// TIA Portal V17 export
// export: Created 2025-03-05T08:00:07.6306461Z, ExportSetting WithDefaults, DisplayName Totally Integrated Automation Portal, DisplayVersion V17 Update 8, DisplayName TIA Portal Openness, DisplayVersion V17 Update 8, DisplayName TIA Portal Version Control Interface, DisplayVersion V17, DisplayName SINAMICS Startdrive Advanced, DisplayVersion V17 SP2, DisplayName SINAMICS Startdrive G110M, G120, G120C, G120D, G120P, G115D, DisplayVersion V17 SP2, DisplayName SINAMICS Startdrive G130, G150, S120, S150, SINAMICS MV, S210, DisplayVersion V17 SP2, DisplayName STEP 7 Professional, DisplayVersion V17 Update 8, DisplayName SINUMERIK ONE STEP 7 Toolbox, DisplayVersion V17 Update 12, DisplayName SINUMERIK 840D sl STEP 7 Toolbox, DisplayVersion V17 Update 12, DisplayName STEP 7 Safety, DisplayVersion V17 Update 6, DisplayName WinCC Advanced, DisplayVersion V17 Update 8
DATA_BLOCK "DB2031_CYCLES_GENERAL"   // DB2031
{ S7_Optimized_Access := 'FALSE'; DB_Accessible_From_OPC_UA := 'FALSE' }
AUTHOR : ETXETAR
VERSION : 1.0
// stored: AutoNumber false, DBAccessibleFromOPCUA false, DBAccessibleFromWebserver true, IsOnlyStoredInLoadMemory false, IsWriteProtectedInAS false
   VAR RETAIN
      CONTINUOUS_CYCLE { S7_SetPoint := 'True'} : "CYCLES";
      SINGLE_CYCLE { S7_SetPoint := 'True'} : "CYCLES";
      RUN_OUT { S7_SetPoint := 'True'} : "CYCLES";
      DRY_CYCLE { S7_SetPoint := 'True'} : "CYCLES";
      MANUAL_LOAD_CYCLE { S7_SetPoint := 'True'} : "CYCLES";
      GANTRY_ROBOT_TEST_CYCLE { S7_SetPoint := 'True'} : "CYCLES";
      GANTRY_DRY_CYCLE { S7_SetPoint := 'True'} : "CYCLES";
      ROBOT_DRY_CYCLE { S7_SetPoint := 'True'} : "CYCLES";
      CALIBRATION_CYCLE { S7_SetPoint := 'True'} : "CYCLES";
      RUN_OUT_UNIT_01 { S7_SetPoint := 'True'} : "CYCLES";
      RUN_OUT_UNIT_02 { S7_SetPoint := 'True'} : "CYCLES";
      MASTER_MEASUREMENT { S7_SetPoint := 'True'} : "CYCLES";
   END_VAR
BEGIN
   CONTINUOUS_CYCLE.GENERAL_CONDITIONS := FALSE;
   CONTINUOUS_CYCLE.INITIAL_CONDITIONS := FALSE;
   CONTINUOUS_CYCLE.ENABLE_REQUEST := FALSE;
   CONTINUOUS_CYCLE.DISABLE_REQUEST := FALSE;
   CONTINUOUS_CYCLE.TOGGLE_COMMAND_P := FALSE;
   CONTINUOUS_CYCLE.WARNING_GONE := FALSE;
   CONTINUOUS_CYCLE.GENERAL_CONDITIONS_HELP := FALSE;
   CONTINUOUS_CYCLE.INITIAL_CONDITIONS_HELP := FALSE;
   CONTINUOUS_CYCLE.CYCLE_SELECTED := FALSE;   // CONTINUOUS CYCLE SELECTED
   CONTINUOUS_CYCLE.CYCLE_SELECTED_AUX := FALSE;
   CONTINUOUS_CYCLE.CYCLE_COMPLETED := FALSE;   // CONTINUOUS CYCLE COMPLETED
   CONTINUOUS_CYCLE.MACHINE_EMPTY := FALSE;
   CONTINUOUS_CYCLE.MACHINE_EMPTY_MANUAL_LOAD_SELECTED := FALSE;
   CONTINUOUS_CYCLE.MACHINE_EMPTY_WO_MANUAL_LOAD_SELECTED := FALSE;
   CONTINUOUS_CYCLE.RESET_FULL_DEPTH_DRY_CYCLE_DISABLED := FALSE;
   CONTINUOUS_CYCLE.RESET_FULL_DEPTHS_AUX := FALSE;
   CONTINUOUS_CYCLE.CYCLE_SEOC := FALSE;
   CONTINUOUS_CYCLE.CYCLE_IS := FALSE;
   SINGLE_CYCLE.GENERAL_CONDITIONS := TRUE;
   SINGLE_CYCLE.INITIAL_CONDITIONS := TRUE;
   SINGLE_CYCLE.ENABLE_REQUEST := FALSE;
   SINGLE_CYCLE.DISABLE_REQUEST := TRUE;
   SINGLE_CYCLE.TOGGLE_COMMAND_P := FALSE;
   SINGLE_CYCLE.WARNING_GONE := FALSE;
   SINGLE_CYCLE.GENERAL_CONDITIONS_HELP := FALSE;
   SINGLE_CYCLE.INITIAL_CONDITIONS_HELP := FALSE;
   SINGLE_CYCLE.CYCLE_SELECTED := FALSE;   // SINGLE CYCLE SELECTED
   SINGLE_CYCLE.CYCLE_SELECTED_AUX := FALSE;
   SINGLE_CYCLE.CYCLE_COMPLETED := FALSE;   // SINGLE CYCLE COMPLETED
   SINGLE_CYCLE.MACHINE_EMPTY := FALSE;
   SINGLE_CYCLE.MACHINE_EMPTY_MANUAL_LOAD_SELECTED := FALSE;
   SINGLE_CYCLE.MACHINE_EMPTY_WO_MANUAL_LOAD_SELECTED := FALSE;
   SINGLE_CYCLE.RESET_FULL_DEPTH_DRY_CYCLE_DISABLED := FALSE;
   SINGLE_CYCLE.RESET_FULL_DEPTHS_AUX := FALSE;
   SINGLE_CYCLE.CYCLE_SEOC := FALSE;
   SINGLE_CYCLE.CYCLE_IS := FALSE;
   RUN_OUT.GENERAL_CONDITIONS := TRUE;
   RUN_OUT.INITIAL_CONDITIONS := TRUE;
   RUN_OUT.ENABLE_REQUEST := FALSE;
   RUN_OUT.DISABLE_REQUEST := FALSE;
   RUN_OUT.TOGGLE_COMMAND_P := FALSE;
   RUN_OUT.WARNING_GONE := FALSE;
   RUN_OUT.GENERAL_CONDITIONS_HELP := FALSE;
   RUN_OUT.INITIAL_CONDITIONS_HELP := FALSE;
   RUN_OUT.CYCLE_SELECTED := FALSE;   // RUN OUT CYCLE SELECTED
   RUN_OUT.CYCLE_SELECTED_AUX := FALSE;
   RUN_OUT.CYCLE_COMPLETED := FALSE;   // RUN OUT CYCLE COMPLETED
   RUN_OUT.MACHINE_EMPTY := FALSE;
   RUN_OUT.MACHINE_EMPTY_MANUAL_LOAD_SELECTED := FALSE;
   RUN_OUT.MACHINE_EMPTY_WO_MANUAL_LOAD_SELECTED := FALSE;
   RUN_OUT.RESET_FULL_DEPTH_DRY_CYCLE_DISABLED := FALSE;
   RUN_OUT.RESET_FULL_DEPTHS_AUX := FALSE;
   RUN_OUT.CYCLE_SEOC := FALSE;
   RUN_OUT.CYCLE_IS := FALSE;
   DRY_CYCLE.GENERAL_CONDITIONS := FALSE;
   DRY_CYCLE.INITIAL_CONDITIONS := FALSE;
   DRY_CYCLE.ENABLE_REQUEST := FALSE;
   DRY_CYCLE.DISABLE_REQUEST := FALSE;
   DRY_CYCLE.TOGGLE_COMMAND_P := FALSE;
   DRY_CYCLE.WARNING_GONE := FALSE;
   DRY_CYCLE.GENERAL_CONDITIONS_HELP := FALSE;
   DRY_CYCLE.INITIAL_CONDITIONS_HELP := FALSE;
   DRY_CYCLE.CYCLE_SELECTED := FALSE;   // DRY CYCLE SELECTED
   DRY_CYCLE.CYCLE_SELECTED_AUX := FALSE;
   DRY_CYCLE.CYCLE_COMPLETED := FALSE;   // DRY CYCLE COMPLETED
   DRY_CYCLE.MACHINE_EMPTY := FALSE;
   DRY_CYCLE.MACHINE_EMPTY_MANUAL_LOAD_SELECTED := FALSE;
   DRY_CYCLE.MACHINE_EMPTY_WO_MANUAL_LOAD_SELECTED := FALSE;
   DRY_CYCLE.RESET_FULL_DEPTH_DRY_CYCLE_DISABLED := FALSE;
   DRY_CYCLE.RESET_FULL_DEPTHS_AUX := FALSE;
   DRY_CYCLE.CYCLE_SEOC := FALSE;
   DRY_CYCLE.CYCLE_IS := FALSE;
   MANUAL_LOAD_CYCLE.GENERAL_CONDITIONS := FALSE;
   MANUAL_LOAD_CYCLE.INITIAL_CONDITIONS := TRUE;
   MANUAL_LOAD_CYCLE.ENABLE_REQUEST := FALSE;
   MANUAL_LOAD_CYCLE.DISABLE_REQUEST := FALSE;
   MANUAL_LOAD_CYCLE.TOGGLE_COMMAND_P := FALSE;
   MANUAL_LOAD_CYCLE.WARNING_GONE := TRUE;
   MANUAL_LOAD_CYCLE.GENERAL_CONDITIONS_HELP := FALSE;
   MANUAL_LOAD_CYCLE.INITIAL_CONDITIONS_HELP := FALSE;
   MANUAL_LOAD_CYCLE.CYCLE_SELECTED := TRUE;   // MANUAL LOAD CYCLE SELECTED
   MANUAL_LOAD_CYCLE.CYCLE_SELECTED_AUX := FALSE;
   MANUAL_LOAD_CYCLE.CYCLE_COMPLETED := FALSE;   // MANUAL LOAD CYCLE COMPLETED
   MANUAL_LOAD_CYCLE.MACHINE_EMPTY := FALSE;
   MANUAL_LOAD_CYCLE.MACHINE_EMPTY_MANUAL_LOAD_SELECTED := FALSE;
   MANUAL_LOAD_CYCLE.MACHINE_EMPTY_WO_MANUAL_LOAD_SELECTED := FALSE;
   MANUAL_LOAD_CYCLE.RESET_FULL_DEPTH_DRY_CYCLE_DISABLED := FALSE;
   MANUAL_LOAD_CYCLE.RESET_FULL_DEPTHS_AUX := FALSE;
   MANUAL_LOAD_CYCLE.CYCLE_SEOC := FALSE;
   MANUAL_LOAD_CYCLE.CYCLE_IS := FALSE;
   GANTRY_ROBOT_TEST_CYCLE.GENERAL_CONDITIONS := FALSE;
   GANTRY_ROBOT_TEST_CYCLE.INITIAL_CONDITIONS := FALSE;
   GANTRY_ROBOT_TEST_CYCLE.ENABLE_REQUEST := FALSE;
   GANTRY_ROBOT_TEST_CYCLE.DISABLE_REQUEST := FALSE;
   GANTRY_ROBOT_TEST_CYCLE.TOGGLE_COMMAND_P := FALSE;
   GANTRY_ROBOT_TEST_CYCLE.WARNING_GONE := FALSE;
   GANTRY_ROBOT_TEST_CYCLE.GENERAL_CONDITIONS_HELP := FALSE;
   GANTRY_ROBOT_TEST_CYCLE.INITIAL_CONDITIONS_HELP := FALSE;
   GANTRY_ROBOT_TEST_CYCLE.CYCLE_SELECTED := FALSE;   // GANTRY ROBOT TEST CYCLE SELECTED
   GANTRY_ROBOT_TEST_CYCLE.CYCLE_SELECTED_AUX := FALSE;
   GANTRY_ROBOT_TEST_CYCLE.CYCLE_COMPLETED := FALSE;   // GANTRY ROBOT TEST CYCLE COMPLETED
   GANTRY_ROBOT_TEST_CYCLE.MACHINE_EMPTY := FALSE;
   GANTRY_ROBOT_TEST_CYCLE.MACHINE_EMPTY_MANUAL_LOAD_SELECTED := FALSE;
   GANTRY_ROBOT_TEST_CYCLE.MACHINE_EMPTY_WO_MANUAL_LOAD_SELECTED := FALSE;
   GANTRY_ROBOT_TEST_CYCLE.RESET_FULL_DEPTH_DRY_CYCLE_DISABLED := FALSE;
   GANTRY_ROBOT_TEST_CYCLE.RESET_FULL_DEPTHS_AUX := FALSE;
   GANTRY_ROBOT_TEST_CYCLE.CYCLE_SEOC := FALSE;
   GANTRY_ROBOT_TEST_CYCLE.CYCLE_IS := FALSE;
   GANTRY_DRY_CYCLE.GENERAL_CONDITIONS := FALSE;
   GANTRY_DRY_CYCLE.INITIAL_CONDITIONS := FALSE;
   GANTRY_DRY_CYCLE.ENABLE_REQUEST := FALSE;
   GANTRY_DRY_CYCLE.DISABLE_REQUEST := FALSE;
   GANTRY_DRY_CYCLE.TOGGLE_COMMAND_P := FALSE;
   GANTRY_DRY_CYCLE.WARNING_GONE := FALSE;
   GANTRY_DRY_CYCLE.GENERAL_CONDITIONS_HELP := FALSE;
   GANTRY_DRY_CYCLE.INITIAL_CONDITIONS_HELP := FALSE;
   GANTRY_DRY_CYCLE.CYCLE_SELECTED := FALSE;   // GANTRY DRY CYCLE SELECTED
   GANTRY_DRY_CYCLE.CYCLE_SELECTED_AUX := FALSE;
   GANTRY_DRY_CYCLE.CYCLE_COMPLETED := FALSE;   // GANTRY DRY CYCLE COMPLETED
   GANTRY_DRY_CYCLE.MACHINE_EMPTY := FALSE;
   GANTRY_DRY_CYCLE.MACHINE_EMPTY_MANUAL_LOAD_SELECTED := FALSE;
   GANTRY_DRY_CYCLE.MACHINE_EMPTY_WO_MANUAL_LOAD_SELECTED := FALSE;
   GANTRY_DRY_CYCLE.RESET_FULL_DEPTH_DRY_CYCLE_DISABLED := FALSE;
   GANTRY_DRY_CYCLE.RESET_FULL_DEPTHS_AUX := FALSE;
   GANTRY_DRY_CYCLE.CYCLE_SEOC := FALSE;
   GANTRY_DRY_CYCLE.CYCLE_IS := FALSE;
   ROBOT_DRY_CYCLE.GENERAL_CONDITIONS := FALSE;
   ROBOT_DRY_CYCLE.INITIAL_CONDITIONS := FALSE;
   ROBOT_DRY_CYCLE.ENABLE_REQUEST := FALSE;
   ROBOT_DRY_CYCLE.DISABLE_REQUEST := FALSE;
   ROBOT_DRY_CYCLE.TOGGLE_COMMAND_P := FALSE;
   ROBOT_DRY_CYCLE.WARNING_GONE := FALSE;
   ROBOT_DRY_CYCLE.GENERAL_CONDITIONS_HELP := FALSE;
   ROBOT_DRY_CYCLE.INITIAL_CONDITIONS_HELP := FALSE;
   ROBOT_DRY_CYCLE.CYCLE_SELECTED := FALSE;   // ROBOT DRY CYCLE SELECTED
   ROBOT_DRY_CYCLE.CYCLE_SELECTED_AUX := FALSE;
   ROBOT_DRY_CYCLE.CYCLE_COMPLETED := FALSE;   // ROBOT DRY CYCLE COMPLETED
   ROBOT_DRY_CYCLE.MACHINE_EMPTY := FALSE;
   ROBOT_DRY_CYCLE.MACHINE_EMPTY_MANUAL_LOAD_SELECTED := FALSE;
   ROBOT_DRY_CYCLE.MACHINE_EMPTY_WO_MANUAL_LOAD_SELECTED := FALSE;
   ROBOT_DRY_CYCLE.RESET_FULL_DEPTH_DRY_CYCLE_DISABLED := FALSE;
   ROBOT_DRY_CYCLE.RESET_FULL_DEPTHS_AUX := FALSE;
   ROBOT_DRY_CYCLE.CYCLE_SEOC := FALSE;
   ROBOT_DRY_CYCLE.CYCLE_IS := FALSE;
END_DATA_BLOCK
